// TIA Portal project "Project1" (V17)

(* hardware
DEVICE "S7-1200 station_1"  S7-1200 Station
   slot 0: "Rack_0"  S7-1200 Rack  Rack  V1.0
   slot 1: "PLC_1"  CPU 1214C DC/DC/DC  6ES7 214-1AG40-0XB0  V4.3
   slot 2: "DI 16x24VDC_1"  6ES7 221-1BH32-0XB0  V2.0
   slot 3: "DQ 16x24VDC_1"  SM 1222 DQ16 x 24VDC  6ES7 222-1BH32-0XB0  V2.0
*)

// ===== PLC "PLC_1"  CPU 1214C DC/DC/DC =====

VAR_GLOBAL   // PLC tag table "Default tag table"
   "Tag_1" AT %M0.0 : Bool;
   "Tag_2" AT %Q0.1 : Bool;
   "Tag_3" AT %I0.0 : Bool;
   "Tag_4" AT %M0.1 : Bool;
END_VAR

// folder: System blocks/Program resources

DATA_BLOCK "IEC_Timer_0_DB"   // DB1
{ S7_Optimized_Access := 'TRUE' }
AUTHOR : Simatic
FAMILY : IEC
NAME : IEC_TMR
VERSION : 1.0
// stored: InstanceOfName IEC_TIMER
"IEC_TIMER"
BEGIN
END_DATA_BLOCK

// folder: (top level)

ORGANIZATION_BLOCK "Main"   // OB1, LAD, ProgramCycle
TITLE = "Main Program Sweep (Cycle)"
{ S7_Optimized_Access := 'TRUE' }
VERSION : 0.1
   VAR_INPUT
      Initial_Call : Bool;   // Initial call of this OB
      Remanence : Bool;   // =True, if remanent data are available
   END_VAR
BEGIN

REGION Network 1
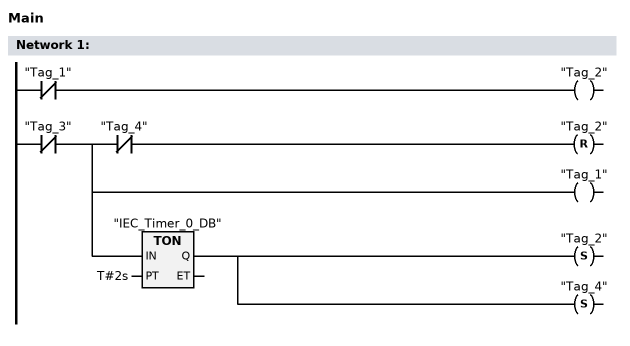
   "Tag_2" := NOT "Tag_1";
   IF NOT "Tag_3" AND NOT "Tag_4" THEN "Tag_2" := FALSE; END_IF;
   "Tag_1" := NOT "Tag_3";
   "IEC_Timer_0_DB".TON(IN := NOT "Tag_3", PT := T#2s);
   IF "IEC_Timer_0_DB".Q THEN
       "Tag_2" := TRUE;
       "Tag_4" := TRUE;
   END_IF;
END_REGION
END_ORGANIZATION_BLOCK